// TIA Portal V17 export
// export: Created 2023-02-13T11:16:00.8108553Z, ExportSetting WithDefaults, DisplayName Totally Integrated Automation Portal, DisplayVersion V17, DisplayName TIA Portal Openness, DisplayVersion V17, DisplayName TIA Portal Teamcenter Gateway, DisplayVersion V17, DisplayName TIA Portal Version Control Interface, DisplayVersion V17, DisplayName SINAMICS Startdrive Advanced, DisplayVersion V17, DisplayName SINAMICS Startdrive G130, G150, S120, S150, SINAMICS MV, S210, DisplayVersion V17, DisplayName SINAMICS Startdrive G110M, G120, G120C, G120D, G120P, G115D, DisplayVersion V17, DisplayName STEP 7 Professional, DisplayVersion V17, DisplayName STEP 7 Safety, DisplayVersion V17, DisplayName WinCC Professional, DisplayVersion V17
FUNCTION_BLOCK "InletWater"   // FB30, LAD
{ S7_Optimized_Access := 'TRUE' }
VERSION : 0.1
// stored: AutoNumber false, IsIECCheckEnabled false, IsRetainMemResEnabled false, MemoryReserve 100, SetENOAutomatically false, UDAEnableTagReadback false
   VAR_INPUT
      IN_FBAV_ProWater : Bool;
      IN_FBAV_HotWater : Bool;
      IN_FBAV_HWT : Bool;
      IN_FT_01 : Real;
      IN_FT_02 : Real;
      IN_FB_PumpHWT : Bool;
   END_VAR
   VAR_OUTPUT
      Q_AV_ProWater : Bool;
      Q_AV_HotWater : Bool;
      Q_PumpHWT : Bool;
   END_VAR
   VAR
      alwaysON : Bool;
      Cmd : Struct
         Pro_Start_Process : Bool;
         Hot_Start_Process : Bool;
         Stop_Process : Bool;
         Reset : Bool;
      END_STRUCT;
      Parameter : Struct
         SP_Prowater : Real;
         SP_Hotwater : Real;
      END_STRUCT;
      State : Struct
         Tank : Struct
            ProWater : Struct
               Idle : Bool;
               Ready_for_Inlet : Bool;
               OnGoing : Bool;
               Error : Bool;
               Done : Bool;
            END_STRUCT;
            HotWater : Struct
               Idle : Bool;
               Ready_for_Inlet : Bool;
               OnGoing : Bool;
               Error : Bool;
               Done : Bool;
            END_STRUCT;
            Status : USInt;
         END_STRUCT;
         HW_Error : Bool;
         Inlet_Done : Bool;
      END_STRUCT;
      Actuator : Struct
         AV_ProWater : Bool;
         AV_HotWater : Bool;
         Pump_HWT : Bool;
      END_STRUCT;
      "Timer" : Struct
         HotWater : IEC_TIMER;
         AVHotWater { S7_SetPoint := 'True'} : IEC_TIMER;
      END_STRUCT;
      N_InletProOnGoing : Bool;
      N_InletHotOnGoing : Bool;
      N_PumpHWT : Bool;
      P_InletProDone : Bool;
      P_InletHotDone : Bool;
      P_Stop : Bool;
      P_Reset : Bool;
      P_InletProReady : Bool;
      N_InletOnGoing : Bool;
   END_VAR
   VAR_TEMP   // added for the SCL form of the ladder/FBD networks
      _w1 : Bool;
      _w2 : Bool;
   END_VAR
BEGIN

REGION Network 1: Always ON
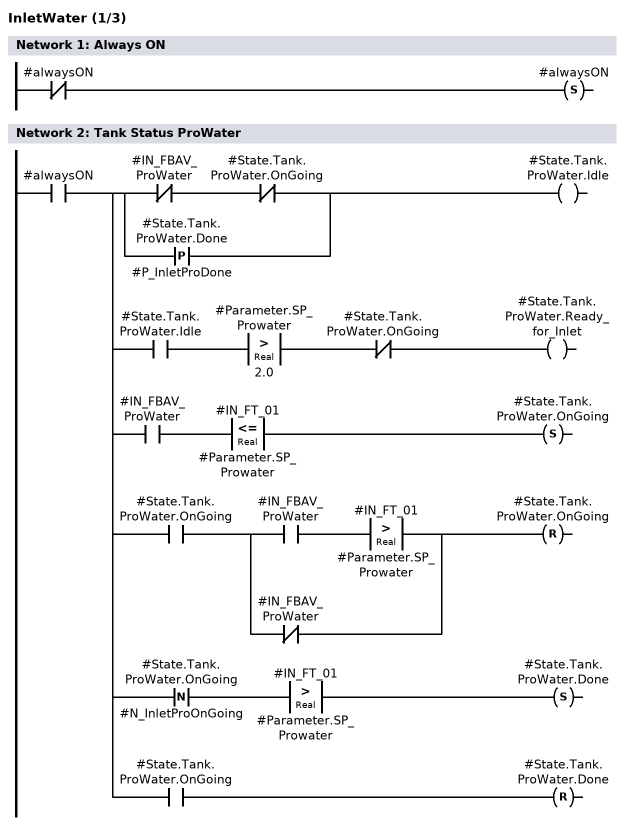
   RUNG wire#powerrail
      I_Contact( #alwaysON )
      S_Coil( #alwaysON )
   END_RUNG
   // the same network as SCL:
   IF NOT #alwaysON THEN #alwaysON := TRUE; END_IF;
END_REGION

REGION Network 2: Tank Status ProWater
   RUNG wire#powerrail
      Contact( #alwaysON )
      wire#w1
      I_Contact( #IN_FBAV_ProWater )
      I_Contact( #State.Tank.ProWater.OnGoing )
      wire#w2
      Coil( #State.Tank.ProWater.Idle )
   END_RUNG
   RUNG wire#w1
      P_Contact(operand := #State.Tank.ProWater.Done, bit := #P_InletProDone)
   END_RUNG wire#w2
   RUNG wire#w1
      Contact( #State.Tank.ProWater.Idle )
      { S7_Templates := "SrcType := Real" } GT_Contact(in1 := #Parameter.SP_Prowater, in2 := 2.0)
      I_Contact( #State.Tank.ProWater.OnGoing )
      Coil( #State.Tank.ProWater.Ready_for_Inlet )
   END_RUNG
   RUNG wire#w1
      Contact( #IN_FBAV_ProWater )
      { S7_Templates := "SrcType := Real" } LE_Contact(in1 := #IN_FT_01, in2 := #Parameter.SP_Prowater)
      S_Coil( #State.Tank.ProWater.OnGoing )
   END_RUNG
   RUNG wire#w1
      Contact( #State.Tank.ProWater.OnGoing )
      wire#w3
      Contact( #IN_FBAV_ProWater )
      { S7_Templates := "SrcType := Real" } GT_Contact(in1 := #IN_FT_01, in2 := #Parameter.SP_Prowater)
      wire#w4
      R_Coil( #State.Tank.ProWater.OnGoing )
   END_RUNG
   RUNG wire#w3
      I_Contact( #IN_FBAV_ProWater )
   END_RUNG wire#w4
   RUNG wire#w1
      N_Contact(operand := #State.Tank.ProWater.OnGoing, bit := #N_InletProOnGoing)
      { S7_Templates := "SrcType := Real" } GT_Contact(in1 := #IN_FT_01, in2 := #Parameter.SP_Prowater)
      S_Coil( #State.Tank.ProWater.Done )
   END_RUNG
   RUNG wire#w1
      Contact( #State.Tank.ProWater.OnGoing )
      R_Coil( #State.Tank.ProWater.Done )
   END_RUNG
   // the same network as SCL:
   #_w1 := #alwaysON AND #State.Tank.ProWater.Done AND NOT #P_InletProDone;   // rising edge of #State.Tank.ProWater.Done
   #P_InletProDone := #State.Tank.ProWater.Done;
   #State.Tank.ProWater.Idle := (#alwaysON AND NOT #IN_FBAV_ProWater AND NOT #State.Tank.ProWater.OnGoing) OR #_w1;
   #State.Tank.ProWater.Ready_for_Inlet := #alwaysON AND #State.Tank.ProWater.Idle AND (#Parameter.SP_Prowater > 2.0) AND NOT #State.Tank.ProWater.OnGoing;
   IF #alwaysON AND #IN_FBAV_ProWater AND (#IN_FT_01 <= #Parameter.SP_Prowater) THEN
       #State.Tank.ProWater.OnGoing := TRUE;
   END_IF;
   IF #alwaysON AND #State.Tank.ProWater.OnGoing AND ((#IN_FBAV_ProWater AND (#IN_FT_01 > #Parameter.SP_Prowater)) OR NOT #IN_FBAV_ProWater) THEN
       #State.Tank.ProWater.OnGoing := FALSE;
   END_IF;
   #_w2 := #alwaysON AND NOT #State.Tank.ProWater.OnGoing AND #N_InletProOnGoing;   // falling edge of #State.Tank.ProWater.OnGoing
   #N_InletProOnGoing := #State.Tank.ProWater.OnGoing;
   IF #_w2 AND (#IN_FT_01 > #Parameter.SP_Prowater) THEN #State.Tank.ProWater.Done := TRUE; END_IF;
   IF #alwaysON AND #State.Tank.ProWater.OnGoing THEN #State.Tank.ProWater.Done := FALSE; END_IF;
END_REGION

REGION Network 3: Tank Status HotWater
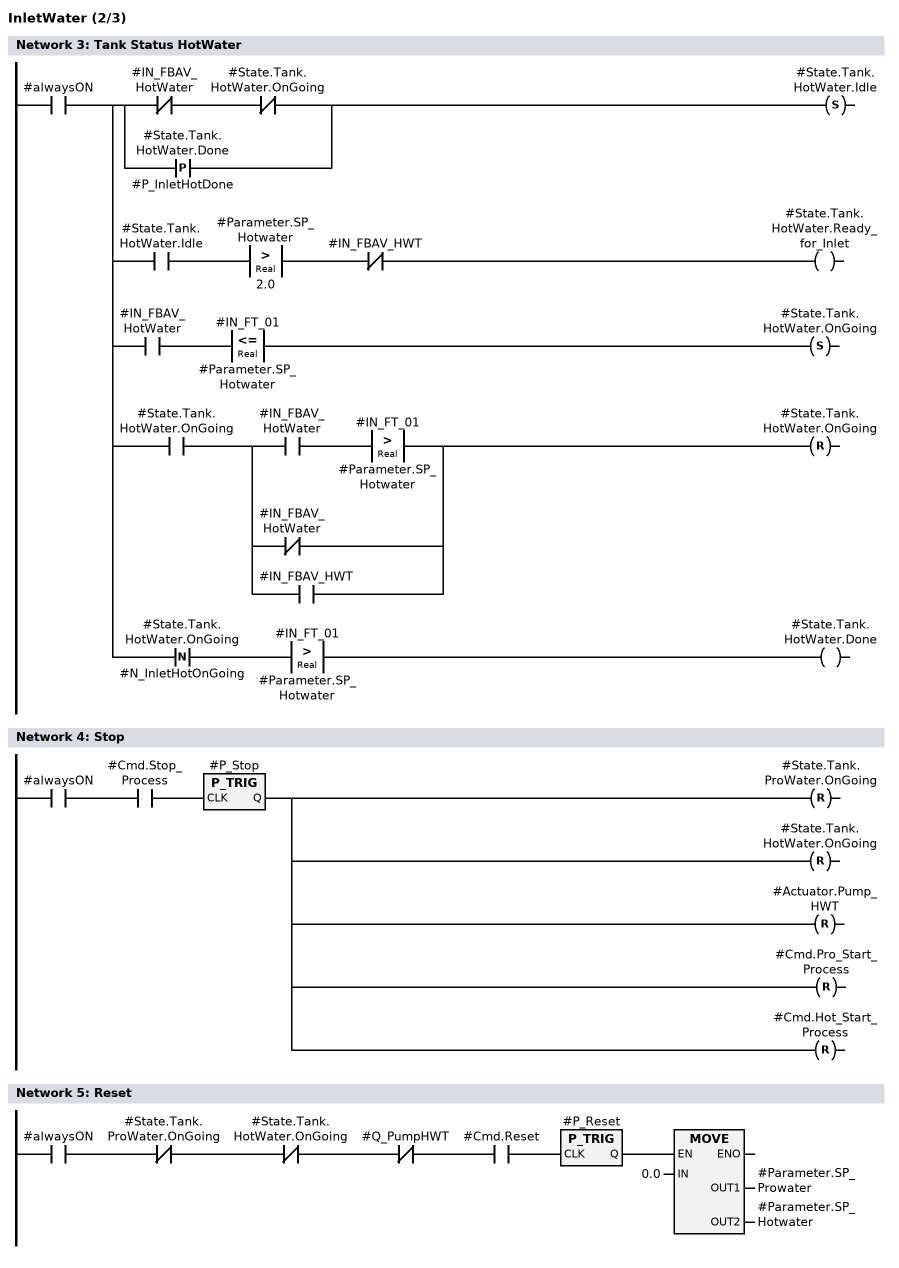
   RUNG wire#powerrail
      Contact( #alwaysON )
      wire#w1
      I_Contact( #IN_FBAV_HotWater )
      I_Contact( #State.Tank.HotWater.OnGoing )
      wire#w2
      S_Coil( #State.Tank.HotWater.Idle )
   END_RUNG
   RUNG wire#w1
      P_Contact(operand := #State.Tank.HotWater.Done, bit := #P_InletHotDone)
   END_RUNG wire#w2
   RUNG wire#w1
      Contact( #State.Tank.HotWater.Idle )
      { S7_Templates := "SrcType := Real" } GT_Contact(in1 := #Parameter.SP_Hotwater, in2 := 2.0)
      I_Contact( #IN_FBAV_HWT )
      Coil( #State.Tank.HotWater.Ready_for_Inlet )
   END_RUNG
   RUNG wire#w1
      Contact( #IN_FBAV_HotWater )
      { S7_Templates := "SrcType := Real" } LE_Contact(in1 := #IN_FT_01, in2 := #Parameter.SP_Hotwater)
      S_Coil( #State.Tank.HotWater.OnGoing )
   END_RUNG
   RUNG wire#w1
      Contact( #State.Tank.HotWater.OnGoing )
      wire#w3
      Contact( #IN_FBAV_HotWater )
      { S7_Templates := "SrcType := Real" } GT_Contact(in1 := #IN_FT_01, in2 := #Parameter.SP_Hotwater)
      wire#w4
      R_Coil( #State.Tank.HotWater.OnGoing )
   END_RUNG
   RUNG wire#w3
      I_Contact( #IN_FBAV_HotWater )
   END_RUNG wire#w4
   RUNG wire#w3
      Contact( #IN_FBAV_HWT )
   END_RUNG wire#w4
   RUNG wire#w1
      N_Contact(operand := #State.Tank.HotWater.OnGoing, bit := #N_InletHotOnGoing)
      { S7_Templates := "SrcType := Real" } GT_Contact(in1 := #IN_FT_01, in2 := #Parameter.SP_Hotwater)
      Coil( #State.Tank.HotWater.Done )
   END_RUNG
   // the same network as SCL:
   #_w1 := #alwaysON AND #State.Tank.HotWater.Done AND NOT #P_InletHotDone;   // rising edge of #State.Tank.HotWater.Done
   #P_InletHotDone := #State.Tank.HotWater.Done;
   IF (#alwaysON AND NOT #IN_FBAV_HotWater AND NOT #State.Tank.HotWater.OnGoing) OR #_w1 THEN
       #State.Tank.HotWater.Idle := TRUE;
   END_IF;
   #State.Tank.HotWater.Ready_for_Inlet := #alwaysON AND #State.Tank.HotWater.Idle AND (#Parameter.SP_Hotwater > 2.0) AND NOT #IN_FBAV_HWT;
   IF #alwaysON AND #IN_FBAV_HotWater AND (#IN_FT_01 <= #Parameter.SP_Hotwater) THEN
       #State.Tank.HotWater.OnGoing := TRUE;
   END_IF;
   IF #alwaysON AND #State.Tank.HotWater.OnGoing AND ((#IN_FBAV_HotWater AND (#IN_FT_01 > #Parameter.SP_Hotwater)) OR NOT #IN_FBAV_HotWater OR #IN_FBAV_HWT) THEN
       #State.Tank.HotWater.OnGoing := FALSE;
   END_IF;
   #_w2 := #alwaysON AND NOT #State.Tank.HotWater.OnGoing AND #N_InletHotOnGoing;   // falling edge of #State.Tank.HotWater.OnGoing
   #N_InletHotOnGoing := #State.Tank.HotWater.OnGoing;
   #State.Tank.HotWater.Done := #_w2 AND (#IN_FT_01 > #Parameter.SP_Hotwater);
END_REGION

REGION Network 4: Stop
   RUNG wire#powerrail
      Contact( #alwaysON )
      Contact( #Cmd.Stop_Process )
      P_Trig( #P_Stop )
      wire#w1
      R_Coil( #State.Tank.ProWater.OnGoing )
   END_RUNG
   RUNG wire#w1
      R_Coil( #State.Tank.HotWater.OnGoing )
   END_RUNG
   RUNG wire#w1
      R_Coil( #Actuator.Pump_HWT )
   END_RUNG
   RUNG wire#w1
      R_Coil( #Cmd.Pro_Start_Process )
   END_RUNG
   RUNG wire#w1
      R_Coil( #Cmd.Hot_Start_Process )
   END_RUNG
   // the same network as SCL:
   #_w1 := #alwaysON AND #Cmd.Stop_Process;
   #_w2 := #_w1 AND NOT #P_Stop;   // rising edge
   #P_Stop := #_w1;
   IF #_w2 THEN
       #State.Tank.ProWater.OnGoing := FALSE;
       #State.Tank.HotWater.OnGoing := FALSE;
       #Actuator.Pump_HWT := FALSE;
       #Cmd.Pro_Start_Process := FALSE;
       #Cmd.Hot_Start_Process := FALSE;
   END_IF;
END_REGION

REGION Network 5: Reset
   RUNG wire#powerrail
      Contact( #alwaysON )
      I_Contact( #State.Tank.ProWater.OnGoing )
      I_Contact( #State.Tank.HotWater.OnGoing )
      I_Contact( #Q_PumpHWT )
      Contact( #Cmd.Reset )
      P_Trig( #P_Reset )
      Move(in := 0.0, out1 => #Parameter.SP_Prowater, out2 => #Parameter.SP_Hotwater)
   END_RUNG
   // the same network as SCL:
   #_w1 := #alwaysON AND NOT #State.Tank.ProWater.OnGoing AND NOT #State.Tank.HotWater.OnGoing AND NOT #Q_PumpHWT AND #Cmd.Reset;
   #_w2 := #_w1 AND NOT #P_Reset;   // rising edge
   #P_Reset := #_w1;
   IF #_w2 THEN
       #Parameter.SP_Prowater := 0.0;
       #Parameter.SP_Hotwater := 0.0;
   END_IF;
END_REGION

REGION Network 6: Inlet ProWater
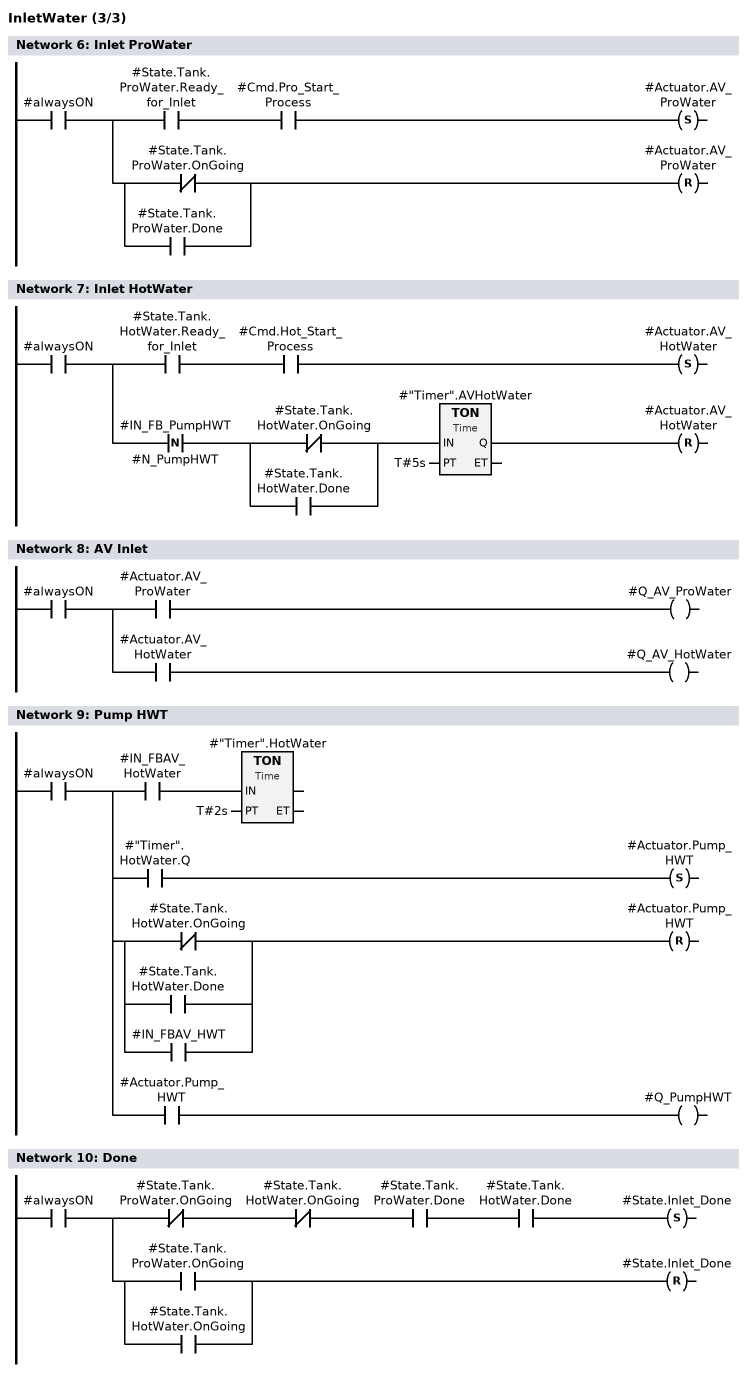
   RUNG wire#powerrail
      Contact( #alwaysON )
      wire#w1
      Contact( #State.Tank.ProWater.Ready_for_Inlet )
      Contact( #Cmd.Pro_Start_Process )
      S_Coil( #Actuator.AV_ProWater )
   END_RUNG
   RUNG wire#w1
      I_Contact( #State.Tank.ProWater.OnGoing )
      wire#w2
      R_Coil( #Actuator.AV_ProWater )
   END_RUNG
   RUNG wire#w1
      Contact( #State.Tank.ProWater.Done )
   END_RUNG wire#w2
   // the same network as SCL:
   IF #alwaysON AND #State.Tank.ProWater.Ready_for_Inlet AND #Cmd.Pro_Start_Process THEN
       #Actuator.AV_ProWater := TRUE;
   END_IF;
   IF #alwaysON AND (NOT #State.Tank.ProWater.OnGoing OR #State.Tank.ProWater.Done) THEN
       #Actuator.AV_ProWater := FALSE;
   END_IF;
END_REGION

REGION Network 7: Inlet HotWater
   RUNG wire#powerrail
      Contact( #alwaysON )
      wire#w1
      Contact( #State.Tank.HotWater.Ready_for_Inlet )
      Contact( #Cmd.Hot_Start_Process )
      S_Coil( #Actuator.AV_HotWater )
   END_RUNG
   RUNG wire#w1
      N_Contact(operand := #IN_FB_PumpHWT, bit := #N_PumpHWT)
      wire#w2
      I_Contact( #State.Tank.HotWater.OnGoing )
      wire#w3
      { S7_Templates := "time_type := Time" } #"Timer".AVHotWater.TON(pt := T#5s, et =>)
      R_Coil( #Actuator.AV_HotWater )
   END_RUNG
   RUNG wire#w2
      Contact( #State.Tank.HotWater.Done )
   END_RUNG wire#w3
   // the same network as SCL:
   IF #alwaysON AND #State.Tank.HotWater.Ready_for_Inlet AND #Cmd.Hot_Start_Process THEN
       #Actuator.AV_HotWater := TRUE;
   END_IF;
   #_w1 := #alwaysON AND NOT #IN_FB_PumpHWT AND #N_PumpHWT;   // falling edge of #IN_FB_PumpHWT
   #N_PumpHWT := #IN_FB_PumpHWT;
   #"Timer".AVHotWater.TON(IN := #_w1 AND (NOT #State.Tank.HotWater.OnGoing OR #State.Tank.HotWater.Done),
                           PT := T#5s);
   IF #"Timer".AVHotWater.Q THEN #Actuator.AV_HotWater := FALSE; END_IF;
END_REGION

REGION Network 8: AV Inlet
   RUNG wire#powerrail
      Contact( #alwaysON )
      wire#w1
      Contact( #Actuator.AV_ProWater )
      Coil( #Q_AV_ProWater )
   END_RUNG
   RUNG wire#w1
      Contact( #Actuator.AV_HotWater )
      Coil( #Q_AV_HotWater )
   END_RUNG
   // the same network as SCL:
   #Q_AV_ProWater := #alwaysON AND #Actuator.AV_ProWater;
   #Q_AV_HotWater := #alwaysON AND #Actuator.AV_HotWater;
END_REGION

REGION Network 9: Pump HWT
   RUNG wire#powerrail
      Contact( #alwaysON )
      wire#w1
      Contact( #IN_FBAV_HotWater )
      { S7_Templates := "time_type := Time" } #"Timer".HotWater.TON(pt := T#2s, et =>)
   END_RUNG
   RUNG wire#w1
      Contact( #"Timer".HotWater.Q )
      S_Coil( #Actuator.Pump_HWT )
   END_RUNG
   RUNG wire#w1
      I_Contact( #State.Tank.HotWater.OnGoing )
      wire#w2
      R_Coil( #Actuator.Pump_HWT )
   END_RUNG
   RUNG wire#w1
      Contact( #State.Tank.HotWater.Done )
   END_RUNG wire#w2
   RUNG wire#w1
      Contact( #IN_FBAV_HWT )
   END_RUNG wire#w2
   RUNG wire#w1
      Contact( #Actuator.Pump_HWT )
      Coil( #Q_PumpHWT )
   END_RUNG
   // the same network as SCL:
   #"Timer".HotWater.TON(IN := #alwaysON AND #IN_FBAV_HotWater, PT := T#2s);
   IF #alwaysON AND #"Timer".HotWater.Q THEN #Actuator.Pump_HWT := TRUE; END_IF;
   IF #alwaysON AND (NOT #State.Tank.HotWater.OnGoing OR #State.Tank.HotWater.Done OR #IN_FBAV_HWT) THEN
       #Actuator.Pump_HWT := FALSE;
   END_IF;
   #Q_PumpHWT := #alwaysON AND #Actuator.Pump_HWT;
END_REGION

REGION Network 10: Done
   RUNG wire#powerrail
      Contact( #alwaysON )
      wire#w1
      I_Contact( #State.Tank.ProWater.OnGoing )
      I_Contact( #State.Tank.HotWater.OnGoing )
      Contact( #State.Tank.ProWater.Done )
      Contact( #State.Tank.HotWater.Done )
      S_Coil( #State.Inlet_Done )
   END_RUNG
   RUNG wire#w1
      Contact( #State.Tank.ProWater.OnGoing )
      wire#w2
      R_Coil( #State.Inlet_Done )
   END_RUNG
   RUNG wire#w1
      Contact( #State.Tank.HotWater.OnGoing )
   END_RUNG wire#w2
   // the same network as SCL:
   IF #alwaysON AND NOT #State.Tank.ProWater.OnGoing AND NOT #State.Tank.HotWater.OnGoing AND #State.Tank.ProWater.Done AND #State.Tank.HotWater.Done THEN
       #State.Inlet_Done := TRUE;
   END_IF;
   IF #alwaysON AND (#State.Tank.ProWater.OnGoing OR #State.Tank.HotWater.OnGoing) THEN
       #State.Inlet_Done := FALSE;
   END_IF;
END_REGION
END_FUNCTION_BLOCK
